# EPICS autosave request: IOCs/12id/iocBoot/ioc12ida1/SBDCM_settings.req
$(P)DCM:Offset.VAL

$(P)DCM:C1_2D.VAL
$(P)DCM:C1_2D.DESC
$(P)DCM:C2_2D.VAL
$(P)DCM:C2_2D.DESC

$(P)Z2_Mode.VAL
$(P)DCM:E2P_driveValue.A
$(P)DCM:E2P_driveValue.B
